(* IEC 61131-3 sources: AXOpen/src/components.cognex.vision/app/src, 2 files *)

(* ---- configuration.st ---- *)
CONFIGURATION MyConfiguration
    TASK Main(Interval := T#10ms, Priority := 1);
    PROGRAM P1 WITH Main: MyProgram;

    VAR_GLOBAL
        {#ix-attr:[Container(Layout.Wrap)]}
        {#ix-set:AttributeName = "If counting PLC is alive"}
        {S7.extern=ReadWrite}
        I_am_alive : ULINT;
        {S7.extern=ReadWrite}
        AxoCognexVisionExampleContext : AxoCognexVisionExample.AxoCognexVisionExampleContext;
        {S7.extern=ReadWrite}
        _rtc : AXOpen.S71500.Rtc;
   END_VAR

    //Copy this VAR_GLOBAL section into your configuration file inside your project.
	//Do not change any names, addresses or any another content.
	VAR_GLOBAL
        {S7.extern=ReadWrite}
		HwInputs AT %IB0 : HwInputs;
        {S7.extern=ReadWrite}
		HwOutputs AT %QB0 : HwOutputs;
        {S7.extern=ReadWrite}
		PlcInputs : PlcInputs;
        {S7.extern=ReadWrite}
		PlcOutputs : PlcOutputs;
	END_VAR

END_CONFIGURATION

(* ---- program.st ---- *)
USING AXOpen.Components.Cognex.Vision;

PROGRAM MyProgram
    VAR_EXTERNAL
        sandbox : SandboxContext;
        documentation : DocumentationContext;
        _rtc : AXOpen.S71500.Rtc;
        _rtm : AXOpen.S71500.Rtm;
    END_VAR

    sandbox.InjectRtc(_rtc);
    sandbox.InjectRtm(_rtm);
    sandbox.Run();

    documentation.InjectRtc(_rtc);
    documentation.InjectRtm(_rtm);
    documentation.Run();
END_PROGRAM
